// TIA Portal V20 export
ORGANIZATION_BLOCK "Startup"   // OB1040, LAD, Startup
TITLE = "Complete Restart"
// stored: AutoNumber false, IsIECCheckEnabled true, Namespace Unit1.Em7, SetENOAutomatically true
   VAR_INPUT
      LostRetentive : Bool;   // True if retentive data are lost
      LostRTC : Bool;   // True if date and time are lost
   END_VAR
BEGIN

REGION Network 1 (SCL): Build the Absolut Reference Designator
   // Set the Absoult Reference Designator in the Config DB
   IF LEN(IN := "Unit1.Em7.Config".em.referenceDesignator.parent) <> 0 THEN
       "Unit1.Em7.Config".em.referenceDesignator.combined := CONCAT_WSTRING(IN1 := "Unit1.Em7.Config".em.referenceDesignator.parent, IN2 := WSTRING#'.', IN3 := "Unit1.Em7.Config".em.referenceDesignator.relative);
   ELSE
       "Unit1.Em7.Config".em.referenceDesignator.combined := "Unit1.Em7.Config".em.referenceDesignator.relative;
   END_IF;
END_REGION

REGION Network 2 (SCL): Assign axes data
   // This is an example how to assign axes to DB_ANY in DB Config. If you have axes, assign them here. The Config.axis[] variables will be handed over to the control modules. That enables a flexible programming.
   // Assign axes
   "Unit1.MotionNodes".PLCToMotion.TechnologyObject.Axis.NGKickerZ := "Unit1.Em7.Config".axis[1] := "BA010AZCRDR10_NgKickerAxisZ";
   "Unit1.MotionNodes".PLCToMotion.TechnologyObject.Axis.PassKickerZ := "Unit1.Em7.Config".axis[2] := "BA010AZCRDR11_PassKickerAxisZ";
   "Unit1.MotionNodes".PLCToMotion.TechnologyObject.Axis.CutConveyor := "Unit1.Em7.Config".axis[3] := "BA010AZCRDR12_CutConveyorAxisB";
   "Unit1.MotionNodes".PLCToMotion.TechnologyObject.Axis.NGConveyor := "Unit1.Em7.Config".axis[4] := "BA010AZCRDR13_NgConveyorAxisB";
   "Unit1.MotionNodes".PLCToMotion.TechnologyObject.Axis.Stack1Conveyor := "Unit1.Em7.Config".axis[5] := "BA010AZCRDR14_Stack1ConveyorAxisB";
   "Unit1.MotionNodes".PLCToMotion.TechnologyObject.Axis.Stack2Conveyor := "Unit1.Em7.Config".axis[6] := "BA010AZCRDR15_Stack2ConveyorAxisB";
   //Config.axis[7] := 
   //Config.axis[8] := 
   //Config.axis[9] :=
   "Unit1.MotionNodes".PLCToMotion.TechnologyObject.Axis.ConveyorVirtual := "Unit1.Em7.Config".axis[10] := "BA010AZCR_ConveyorVirtualAxis";

   // Cam
   //Config.cam[1] :=
   //Config.cam[2] :=
   "Unit1.MotionNodes".PLCToMotion.TechnologyObject.Cam.CutConveyorCam := "Unit1.Em7.Config".cam[3] := "BA010AZCRDR12_CutConveyorAxisBCamMain";
   "Unit1.MotionNodes".PLCToMotion.TechnologyObject.Cam.NgConveyorCam := "Unit1.Em7.Config".cam[4] := "BA010AZCRDR13_NgConveyorAxisBCamMain";
   "Unit1.MotionNodes".PLCToMotion.TechnologyObject.Cam.Stack1ConveyorCam := "Unit1.Em7.Config".cam[5] := "BA010AZCRDR14_Stack1ConveyorAxisBCamMain";
   "Unit1.MotionNodes".PLCToMotion.TechnologyObject.Cam.Stack2ConveyorCamMain := "Unit1.Em7.Config".cam[6] := "BA010AZCRDR15_Stack2ConveyorAxisBCamMain";
   "Unit1.MotionNodes".PLCToMotion.TechnologyObject.Cam.Stack2ConveyorCamSub := "Unit1.Em7.Config".cam[7] := "BA010AZCRDR15_Stack2ConveyorAxisBCamSub";
   //Config.cam[8] :=
   //Config.cam[9] :=
   "Unit1.MotionNodes".PLCToMotion.TechnologyObject.Cam.ConveyorVirtualCam := "Unit1.Em7.Config".cam[10] := "BA010AZCR_ConveyorVirtualAxisCamMain";

   // HW_SubModule
   "Unit1.Em7.Config".moduleAccessPoint[1] := "BA010AZCRCU3~BA010AZARCU3_X150~BA010AZCRDR10_ModuleAccessP,,,";
   "Unit1.Em7.Config".moduleAccessPoint[2] := "BA010AZCRCU3~BA010AZARCU3_X150~BA010AZCRDR11_ModuleAccessP,,,";
   "Unit1.Em7.Config".moduleAccessPoint[3] := "BA010AZCRCU3~BA010AZARCU3_X150~BA010AZCRDR12_ModuleAccessP,,,";
   "Unit1.Em7.Config".moduleAccessPoint[4] := "BA010AZCRCU3~BA010AZARCU3_X150~BA010AZCRDR13_ModuleAccessP,,,";
   "Unit1.Em7.Config".moduleAccessPoint[5] := "BA010AZCRCU3~BA010AZARCU3_X150~BA010AZCRDR14_ModuleAccessP,,,";
   "Unit1.Em7.Config".moduleAccessPoint[6] := "BA010AZCRCU3~BA010AZARCU3_X150~BA010AZCRDR15_ModuleAccessP,,,";
   "Unit1.Em7.Config".moduleAccessPoint[7] := "BA010AZCRDR16~PROFINET_interface~Standard_telegram_1";
   "Unit1.Em7.Config".moduleAccessPoint[8] := "BA010AZCRDR17~PROFINET_interface~Standard_telegram_1";
   "Unit1.Em7.Config".moduleAccessPoint[9] := "BA010AZCRDR18~PROFINET_interface~Standard_telegram_1";
   //Config.moduleAccessPoint[10] :=

   // FB Enable
   "Unit1.Em7.HmiInterface".cmConveyorVirtualAxisB.commands.enable := TRUE;
   "Unit1.Em7.HmiInterface".cmNgKickerAxisZ.commands.enable := TRUE;
   "Unit1.Em7.HmiInterface".cmPassKickerAxisZ.commands.enable := TRUE;
   "Unit1.Em7.HmiInterface".cmCutConveyorAxisB.commands.enable := TRUE;
   "Unit1.Em7.HmiInterface".cmNgConveyorAxisB.commands.enable := TRUE;
   "Unit1.Em7.HmiInterface".cmStack1ConveyorAxisB.commands.enable := TRUE;
   "Unit1.Em7.HmiInterface".cmStack2ConveyorAxisB.commands.enable := TRUE;
   "Unit1.Em7.HmiInterface".cmCutConveyorRingBlow.commands.enableControl := TRUE;
   "Unit1.Em7.HmiInterface".cmNgConveyorRingBlow.commands.enableControl := TRUE;
   "Unit1.Em7.HmiInterface".cmStack2ConveyorRingBlow.commands.enableControl := TRUE;

   // Assign configuration Homing
   "Unit1.Em7.ControlNodes".cmNgKickerAxisZ.commandConfiguration.homing.mode := "Unit1.Em7.HmiInterface".cmNgKickerAxisZ.commandConfiguration.homing.mode := 3;
   "Unit1.Em7.ControlNodes".cmPassKickerAxisZ.commandConfiguration.homing.mode := "Unit1.Em7.HmiInterface".cmPassKickerAxisZ.commandConfiguration.homing.mode := 3;
END_REGION

REGION Network 3 (SCL): CM Config
   // Conveyor Virtual Axis
   "Unit1.Em7.Config".cmConveyorVirtualAxisB.referenceDesignator := WSTRING#'Conveyor Line Speed';
   "Unit1.Em7.Config".cmConveyorVirtualAxisB.disableAlarms := FALSE;
   "Unit1.Em7.Config".cmConveyorVirtualAxisB.masterControlPopUp := TRUE;


   // NgG Kicker Axis Z
   "Unit1.Em7.Config".cmNgKickerAxisZ.referenceDesignator := WSTRING#'Ng Kicker Axis Z';
   "Unit1.Em7.Config".cmNgKickerAxisZ.disableAlarms := FALSE;
   "Unit1.Em7.Config".cmNgKickerAxisZ.masterControlPopUp := TRUE;


   // Pass Kicker Axis Z
   "Unit1.Em7.Config".cmPassKickerAxisZ.referenceDesignator := WSTRING#'Pass Kicker Axis Z';
   "Unit1.Em7.Config".cmPassKickerAxisZ.disableAlarms := FALSE;
   "Unit1.Em7.Config".cmPassKickerAxisZ.masterControlPopUp := TRUE;


   // Cut Conveyor Axis B
   "Unit1.Em7.Config".cmCutConveyorAxisB.referenceDesignator := WSTRING#'Cut Conveyor Axis B';
   "Unit1.Em7.Config".cmCutConveyorAxisB.disableAlarms := FALSE;
   "Unit1.Em7.Config".cmCutConveyorAxisB.masterControlPopUp := TRUE;


   // NG Conveyor Axis B
   "Unit1.Em7.Config".cmNgConveyorAxisB.referenceDesignator := WSTRING#'Ng Conveyor Axis B';
   "Unit1.Em7.Config".cmNgConveyorAxisB.disableAlarms := FALSE;
   "Unit1.Em7.Config".cmNgConveyorAxisB.masterControlPopUp := TRUE;


   // Stack1 Conveyor Axis B
   "Unit1.Em7.Config".cmStack1ConveyorAxisB.referenceDesignator := WSTRING#'Stack1 Conveyor Axis B';
   "Unit1.Em7.Config".cmStack1ConveyorAxisB.disableAlarms := FALSE;
   "Unit1.Em7.Config".cmStack1ConveyorAxisB.masterControlPopUp := TRUE;


   // Stack2 Conveyor Axis B
   "Unit1.Em7.Config".cmStack2ConveyorAxisB.referenceDesignator := WSTRING#'Stack2 Conveyor Axis B';
   "Unit1.Em7.Config".cmStack2ConveyorAxisB.disableAlarms := FALSE;
   "Unit1.Em7.Config".cmStack2ConveyorAxisB.masterControlPopUp := TRUE;


   // Cut Conveyor RingBblow
   "Unit1.Em7.Config".cmCutConveyorRingBlow.disableAlarms := FALSE;
   "Unit1.Em7.Config".cmCutConveyorRingBlow.referenceDesignator := WSTRING#'Cut Conveyor Ringblow';
   "Unit1.Em7.Config".cmCutConveyorRingBlow.masterControlPopUp := TRUE;


   // Ng Conveyor RingBblow
   "Unit1.Em7.Config".cmNgConveyorRingBlow.disableAlarms := FALSE;
   "Unit1.Em7.Config".cmNgConveyorRingBlow.referenceDesignator := WSTRING#'NG Conveyor Ringblow';
   "Unit1.Em7.Config".cmNgConveyorRingBlow.masterControlPopUp := TRUE;


   // stack2 Conveyor RingBblow
   "Unit1.Em7.Config".cmStack2ConveyorRingBlow.disableAlarms := FALSE;
   "Unit1.Em7.Config".cmStack2ConveyorRingBlow.referenceDesignator := WSTRING#'Stack2 Conveyor Ringblow';
   "Unit1.Em7.Config".cmStack2ConveyorRingBlow.masterControlPopUp := TRUE;


   // NgG Box Lock Cylinder
   "Unit1.Em7.Config".cmNgBoxLockCylinderUpDown.referenceDesignator := WSTRING#'Ng Box Lock Cylinder';
   "Unit1.Em7.Config".cmNgBoxLockCylinderUpDown.monitoringLeavingFeedback := T#5s;
   "Unit1.Em7.Config".cmNgBoxLockCylinderUpDown.monitoringReachingFeedback := T#5s;
   "Unit1.Em7.Config".cmNgBoxLockCylinderUpDown.monitoringDiscrepancy := T#0ms;
   "Unit1.Em7.Config".cmNgBoxLockCylinderUpDown.setOutputHomeContinuously := TRUE;
   "Unit1.Em7.Config".cmNgBoxLockCylinderUpDown.setOutputWorkContinuously := TRUE;
   "Unit1.Em7.Config".cmNgBoxLockCylinderUpDown.disableHomeCommand := FALSE;
   "Unit1.Em7.Config".cmNgBoxLockCylinderUpDown.disableFeedbackHomePos := FALSE;
   "Unit1.Em7.Config".cmNgBoxLockCylinderUpDown.disableFeedbackWorkPos := FALSE;
   "Unit1.Em7.Config".cmNgBoxLockCylinderUpDown.disableAlarms := FALSE;
   "Unit1.Em7.Config".cmNgBoxLockCylinderUpDown.resetOutputsOnError := FALSE;
   "Unit1.Em7.Config".cmNgBoxLockCylinderUpDown.allwaysWaitOnReachingTime := FALSE;


   // stack1 QR Reader Fix
   "Unit1.Em7.Config".cmStack1QrReader.hwID.handshakeGeneralErrorStatusHwId := "BA010AZCRCAM1~Handshake_and_General_Error_Status_,,,";
   "Unit1.Em7.Config".cmStack1QrReader.hwID.busyStatusHwId := "BA010AZCRCAM1~BUSY_Status_Bits_1";
   "Unit1.Em7.Config".cmStack1QrReader.hwID.completionStatusHwId := "BA010AZCRCAM1~Completion_Status_Bits_1";
   "Unit1.Em7.Config".cmStack1QrReader.hwID.errorStatusHwId := "BA010AZCRCAM1~Error_Status_Bits_1";
   "Unit1.Em7.Config".cmStack1QrReader.hwID.terminalStatusHwId := "BA010AZCRCAM1~Terminal_Status_Bits_1";
   "Unit1.Em7.Config".cmStack1QrReader.hwID.unstableReadStatusHwId := "BA010AZCRCAM1~Unstable_Read_Status_Bits_1";
   "Unit1.Em7.Config".cmStack1QrReader.hwID.matchingAndGradeStatusHwId := "BA010AZCRCAM1~Matching_Level_and_Total_Evaluation,,,";
   "Unit1.Em7.Config".cmStack1QrReader.hwID.operationResultStatusHwId := "BA010AZCRCAM1~Operation_Result_Status_1";
   "Unit1.Em7.Config".cmStack1QrReader.hwID.readDataHeaderHwId := "BA010AZCRCAM1~Read_Data_128Byte_1";
   "Unit1.Em7.Config".cmStack1QrReader.hwID.latchErrorClearControlHwId := "BA010AZCRCAM1~Latch_and_Error_Clear_Control_Bits_1";
   "Unit1.Em7.Config".cmStack1QrReader.hwID.operationInstructionControlHwId := "BA010AZCRCAM1~Operation_instruction_Control_Bits_1";
   "Unit1.Em7.Config".cmStack1QrReader.hwID.completionClearControlHwId := "BA010AZCRCAM1~Completion_Clear_Control_Bits_1";
   "Unit1.Em7.Config".cmStack1QrReader.hwID.parameterBankNumberHwId := "BA010AZCRCAM1~Parameter_Bank_Number_1";
   "Unit1.Em7.Config".cmStack1QrReader.hwID.userDataHwId := "BA010AZCRCAM1~User_Data_128Byte_1";
   "Unit1.Em7.Config".cmStack1QrReader.triggertime := T#50ms;
   "Unit1.Em7.Config".cmStack1QrReader.cycleTime := T#750ms;


   // stack2 QR Reader Fix
   "Unit1.Em7.Config".cmStack2QrReader.hwID.handshakeGeneralErrorStatusHwId := "BA010AZCRCAM2~Handshake_and_General_Error_Status_,,,";
   "Unit1.Em7.Config".cmStack2QrReader.hwID.busyStatusHwId := "BA010AZCRCAM2~BUSY_Status_Bits_1";
   "Unit1.Em7.Config".cmStack2QrReader.hwID.completionStatusHwId := "BA010AZCRCAM2~Completion_Status_Bits_1";
   "Unit1.Em7.Config".cmStack2QrReader.hwID.errorStatusHwId := "BA010AZCRCAM2~Error_Status_Bits_1";
   "Unit1.Em7.Config".cmStack2QrReader.hwID.terminalStatusHwId := "BA010AZCRCAM2~Terminal_Status_Bits_1";
   "Unit1.Em7.Config".cmStack2QrReader.hwID.unstableReadStatusHwId := "BA010AZCRCAM2~Unstable_Read_Status_Bits_1";
   "Unit1.Em7.Config".cmStack2QrReader.hwID.matchingAndGradeStatusHwId := "BA010AZCRCAM2~Matching_Level_and_Total_Evaluation,,,";
   "Unit1.Em7.Config".cmStack2QrReader.hwID.operationResultStatusHwId := "BA010AZCRCAM2~Operation_Result_Status_1";
   "Unit1.Em7.Config".cmStack2QrReader.hwID.readDataHeaderHwId := "BA010AZCRCAM2~Read_Data_128Byte_1";
   "Unit1.Em7.Config".cmStack2QrReader.hwID.latchErrorClearControlHwId := "BA010AZCRCAM2~Latch_and_Error_Clear_Control_Bits_1";
   "Unit1.Em7.Config".cmStack2QrReader.hwID.operationInstructionControlHwId := "BA010AZCRCAM2~Operation_instruction_Control_Bits_1";
   "Unit1.Em7.Config".cmStack2QrReader.hwID.completionClearControlHwId := "BA010AZCRCAM2~Completion_Clear_Control_Bits_1";
   "Unit1.Em7.Config".cmStack2QrReader.hwID.parameterBankNumberHwId := "BA010AZCRCAM2~Parameter_Bank_Number_1";
   "Unit1.Em7.Config".cmStack2QrReader.hwID.userDataHwId := "BA010AZCRCAM2~User_Data_128Byte_1";
   "Unit1.Em7.Config".cmStack2QrReader.triggertime := T#50ms;
   "Unit1.Em7.Config".cmStack2QrReader.cycleTime := T#750ms;


   // NG Box Detect Sensor
   "Unit1.Em7.Config".CmNgBoxDetectSensor.referenceDesignator := WSTRING#'DigitalSignal';
   "Unit1.Em7.Config".CmNgBoxDetectSensor.onDelay := T#0ms;
   "Unit1.Em7.Config".CmNgBoxDetectSensor.offDelay := T#0ms;
   "Unit1.Em7.Config".CmNgBoxDetectSensor.default := FALSE;
   "Unit1.Em7.Config".CmNgBoxDetectSensor.invertProcessValue := FALSE;
   "Unit1.Em7.Config".CmNgBoxDetectSensor.disableAlarms := FALSE;


   // NG Box Full Sensor
   "Unit1.Em7.Config".CmNgBoxFullSensor.referenceDesignator := WSTRING#'DigitalSignal';
   "Unit1.Em7.Config".CmNgBoxFullSensor.onDelay := T#0ms;
   "Unit1.Em7.Config".CmNgBoxFullSensor.offDelay := T#0ms;
   "Unit1.Em7.Config".CmNgBoxFullSensor.default := FALSE;
   "Unit1.Em7.Config".CmNgBoxFullSensor.invertProcessValue := FALSE;
   "Unit1.Em7.Config".CmNgBoxFullSensor.disableAlarms := FALSE;


   // Ng Kicker Detect Sensor
   "Unit1.Em7.Config".CmNgKickerDetectSensor.referenceDesignator := WSTRING#'DigitalSignal';
   "Unit1.Em7.Config".CmNgKickerDetectSensor.onDelay := T#0ms;
   "Unit1.Em7.Config".CmNgKickerDetectSensor.offDelay := T#0ms;
   "Unit1.Em7.Config".CmNgKickerDetectSensor.default := FALSE;
   "Unit1.Em7.Config".CmNgKickerDetectSensor.invertProcessValue := FALSE;
   "Unit1.Em7.Config".CmNgKickerDetectSensor.disableAlarms := FALSE;

   // Pass Kicker Detect Sensor
   "Unit1.Em7.Config".CmPassKickerDetectSensor.referenceDesignator := WSTRING#'DigitalSignal';
   "Unit1.Em7.Config".CmPassKickerDetectSensor.onDelay := T#0ms;
   "Unit1.Em7.Config".CmPassKickerDetectSensor.offDelay := T#0ms;
   "Unit1.Em7.Config".CmPassKickerDetectSensor.default := FALSE;
   "Unit1.Em7.Config".CmPassKickerDetectSensor.invertProcessValue := FALSE;
   "Unit1.Em7.Config".CmPassKickerDetectSensor.disableAlarms := FALSE;

   // Stack1 Conveyor Electrode Detect Sensor
   "Unit1.Em7.Config".CmStack1ConveyorElectrodeDetectSensor.referenceDesignator := WSTRING#'DigitalSignal';
   "Unit1.Em7.Config".CmStack1ConveyorElectrodeDetectSensor.onDelay := T#0ms;
   "Unit1.Em7.Config".CmStack1ConveyorElectrodeDetectSensor.offDelay := T#0ms;
   "Unit1.Em7.Config".CmStack1ConveyorElectrodeDetectSensor.default := FALSE;
   "Unit1.Em7.Config".CmStack1ConveyorElectrodeDetectSensor.invertProcessValue := FALSE;
   "Unit1.Em7.Config".CmStack1ConveyorElectrodeDetectSensor.disableAlarms := FALSE;

   // Stack2 Conveyor Electrode Detect Sensor
   "Unit1.Em7.Config".CmStack2ConveyorElectrodeDetectSensor.referenceDesignator := WSTRING#'DigitalSignal';
   "Unit1.Em7.Config".CmStack2ConveyorElectrodeDetectSensor.onDelay := T#0ms;
   "Unit1.Em7.Config".CmStack2ConveyorElectrodeDetectSensor.offDelay := T#0ms;
   "Unit1.Em7.Config".CmStack2ConveyorElectrodeDetectSensor.default := FALSE;
   "Unit1.Em7.Config".CmStack2ConveyorElectrodeDetectSensor.invertProcessValue := FALSE;
   "Unit1.Em7.Config".CmStack2ConveyorElectrodeDetectSensor.disableAlarms := FALSE;

   // Alarm Count referenceDesignator
   "Unit1.Em7.HmiInterface".ngKickerSensorNotDetectedCount.referenceDesignator := WSTRING#'NG Kicker Sensor Not Detected Count';
   "Unit1.Em7.HmiInterface".passKickerSensorNotDetectedCount.referenceDesignator := WSTRING#'Pass Kicker Sensor Not Detected Count';
   "Unit1.Em7.HmiInterface".stack1ConveyorElectrodeSensorNotDetectedCount.referenceDesignator := WSTRING#'Stack1 CV Electrode Sensor Not Detected Count';
   "Unit1.Em7.HmiInterface".stack2ConveyorElectrodeSensorNotDetectedCount.referenceDesignator := WSTRING#'Stack2 CV Electrode Sensor Not Detected Count';
   "Unit1.Em7.HmiInterface".visionConsecutiveNgOutCount.referenceDesignator := WSTRING#'Vision Consecutive NG Out Count';
END_REGION
END_ORGANIZATION_BLOCK
